{attribute 'qualified_only'}
VAR_GLOBAL
	// udiDI%41.0_A2_5
	HRL_Enc_horizontal_I1 AT %I*: UDINT;
	// udiDI%47.0_A2_5
	HRL_Enc_horizontal_I2 AT %I*: UDINT;
	// udiDI%53.0_A2_5
	HRL_Enc_vertikal_I1 AT %I*: UDINT;
	// udiDI%59.0_A2_5
	HRL_Enc_vertikal_I2 AT %I*: UDINT;
	// xDI%136.0_A2_2
	HRL_Ref_Taster_horizontal AT %I*: BOOL;
	// xDI%136.1_A2_1
	HRL_LS_innen AT %I*: BOOL;
	// xDI%136.2_A2_1
	HRL_LS_aussen AT %I*: BOOL;
	// xDI%136.3_A2_2
	HRL_Ref_Taster_vertikal AT %I*: BOOL;
	// xDI%136.4_A2_3
	HRL_Spursensor_1_unten AT %I*: BOOL;
	// xDI%136.5_A2_3
	HRL_Spursensor_2_oben AT %I*: BOOL;
	// xDI%136.6_A2_2
	HRL_Ref_Taster_Ausleger_vorne AT %I*: BOOL;
	// xDI%136.7_A2_2
	HRL_Ref_Taster_Ausleger_hinten AT %I*: BOOL;
	// xDO%111.0_A2_2	
	HRL_MOT_Foerderband_vorwaerts AT %Q*: BOOL;
	// xDO%111.1_A2_2
	HRL_MOT_Foerderband_rueckwaerts AT %Q*: BOOL;
	// xDO%111.2_A2_4
	HRL_MOT_horizontal_zum_Regal AT %Q*: BOOL;
	// xDO%111.3_A2_4
	HRL_MOT_horizontal_zum_Foerderband AT %Q*: BOOL;
	// xDO%111.4_A2_4
	HRL_MOT_vertikal_runter AT %Q*: BOOL;
	// xDO%111.5_A2_4
	HRL_MOT_vertikal_hoch AT %Q*: BOOL;
	// xDO%111.6_A2_4
	HRL_MOT_Ausleger_vorwaerts AT %Q*: BOOL;
	// xDO%111.7_A2_4
	HRL_MOT_Ausleger_rueckwaerts AT %Q*: BOOL;
	HRL_K1_1_Zaehler_Zuruecksetzen AT %Q*: BOOL;
	HRL_K1_2_Zaehler_Zuruecksetzen AT %Q*: BOOL;
END_VAR

(* stored: Version 1.1.0.1, ProductVersion 3.1.4024.13
   GVL GVL_HRL: Id {60e560c2-6aa7-4ee1-b402-1bce5cb4b604} *)
